{attribute addProperty BoxType "EK1100-0000-0018"}
{attribute addProperty Id "Beckhoff_EM3xxxEK1122Beckhoff_EM3xxxEK1122_34A2240D162A_0001_EM3701_0000_0016EM3701_6ABA943A11414.25A_0002_EM3702_0000_0016EM3702_963644BA14618.25A_0003_EM3712_0000_0016EM3712_963644BA14618.25"}
{attribute addProperty CRC "236652117"}
{attribute addProperty SizeInBites "422"}
{attribute addProperty SizeInBytes "52.75"}
TYPE Beckhoff_EM3xxx_0E1B0655 EXTENDS EK1100_179A0949 :
STRUCT
	{attribute addProperty Name "Beckhoff_EM3xxxEK1122"}
	Beckhoff_EM3xxxEK1122 : Beckhoff_EM3xxxEK1122_34A2240D;
	{attribute addProperty Name "A_0001_EM3701_0000_0016"}
	A_0001_EM3701_0000_0016 : EM3701_6ABA943A;
	{attribute addProperty Name "A_0002_EM3702_0000_0016"}
	A_0002_EM3702_0000_0016 : EM3702_963644BA;
	{attribute addProperty Name "A_0003_EM3712_0000_0016"}
	A_0003_EM3712_0000_0016 : EM3712_963644BA;
END_STRUCT
END_TYPE

(* stored: Version 1.2.0.0, ProductVersion 3.1.4024.9
   DUT Beckhoff_EM3xxx_0E1B0655: Id {f4a949c3-f8a4-407d-a62b-85ec129cb9d1} *)
